{attribute 'qualified_only'}
{attribute 'strict'}
TYPE PD6ControlWord :
(
	Shutdown := 6,					// 2#0000_0110	
	SwitchOn := 7,					// 0xxx 0111 (Trasition from Ready to Switch On -> Switched On)
	SwitchOnOperationEnable := 15,	// 0xxx 1111 (Switch On and Enable Operation)
	StartHoming:= 16,
	PulseInhibit := 0,				// 0xxx xx0x (activate quick stop and disable)
	QuickStop := 2,					// 0xxx x01x
	DisableOperation := 7,			// 0xxx 0111 (Transition from OpEnable -> Switched On)
	EnableOperation := 15,			// 0xxx 1111
	FaultReset := 128,				// 1xxx xxxx
	StartMove := 2#00010000,				// xxx1 1111
	AbsoluteMotion := 2#00100000			// xxx1 1111
	// Positive := 64,					// x1xx xxxx
	// Negative :=	0					// x0xx xxxx
)BYTE;
END_TYPE

(* stored: Version 1.1.0.1, ProductVersion 3.1.4024.12
   DUT PD6ControlWord: Id {6aced678-c962-4eb6-8812-bce088f967da} *)
